(* CoDeSys 2.3.9.50 project: TcNcsample PTPmove.pro *)
(* Libraries: STANDARD.LIB 5.6.98 12:03:02, TcBase.lib 14.5.09 12:14:08, TcSystem.lib 7.6.16 11:01:22, TcNC.lib 10.10.08 17:55:34, TcMC.lib 27.7.15 08:51:38, TcBaseMath.lib 27.7.04 12:07:56, TcMath.lib 23.9.04 15:15:30 *)

(* Task configuration *)
TASK Standard (PRIORITY := 0, INTERVAL := T#10ms);
	MAIN
END_TASK

(* Global variable list: Global_Variables *)
VAR_GLOBAL
	(* =====================================================	*)
	(* NC · cyclical interface								*)
	(* =====================================================	*)

	PlcToNc AT %Q*	: PLCTONC_AXLESTRUCT;
	NcToPlc AT %I*	: NCTOPLC_AXLESTRUCT;
END_VAR

(* Global variable list: TwinCAT_Configuration *)
(* Generated automatically by TwinCAT - (read only) *)
VAR_CONFIG
	.PlcToNc AT %QB0 : PLCTONC_AXLESTRUCT;	(*  ~ {LinkedWith:TINC^NC-Task 1 SAF^Axes^Axis 1^Inputs^Axis 1_FromPlc} *)
	.NcToPlc AT %IB0 : NCTOPLC_AXLESTRUCT;	(*  ~ {LinkedWith:TINC^NC-Task 1 SAF^Axes^Axis 1^Outputs^Axis 1_ToPlc} *)
END_VAR

(* Data type *)
TYPE MoveState_t :
 (
	MOVESTATE_INIT,
	MOVESTATE_FORWARD,
	MOVESTATE_BACKWARDS
 );
END_TYPE

(* POU MAIN, ST *)
PROGRAM MAIN
VAR
	Position: LREAL;
	StartAxis: BOOL;
	MoveAxis: MC_MoveAbsolute;
	MoveDone: BOOL;
	MoveAborted: BOOL;
	MoveError: BOOL;
	MoveErrorID: UDINT;
	state: MoveState_t;
END_VAR
	(* enable the axis *)
	AxisEnable;

	(* 	move the axis forward and backwards
	*)
	CASE state OF
		MOVESTATE_INIT :	(* initialisation *)
			StartAxis := FALSE;
			IF AxisEnable.Ready THEN
				state := MOVESTATE_FORWARD;
			END_IF

		MOVESTATE_FORWARD :	(* start to first position *)
			Position := 2000;
			StartAxis := TRUE;
			IF MoveDone THEN
				StartAxis := FALSE;
				state := MOVESTATE_BACKWARDS;
			END_IF

		MOVESTATE_BACKWARDS :	(* move back to initial position *)
			Position := 0;
			StartAxis := TRUE;
			IF MoveDone THEN
				StartAxis := FALSE;
				state := MOVESTATE_FORWARD;
			END_IF
	END_CASE

	MoveAction;	(* call the move function block *)



	xxxx
	yyyy
zzzzzgit
END_PROGRAM
ACTION MoveAction:
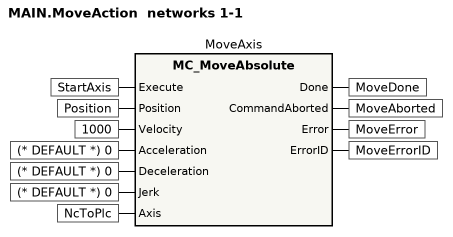
_FBD_ (* Function Block Diagram *)
NETWORK 1 (* Start axis using standard values FOR acceleration, deceleration AND jerk *)
	MoveAxis:MC_MoveAbsolute(Execute: StartAxis, Position: Position, Velocity: 1000, Acceleration: (* DEFAULT *) 0, Deceleration: (* DEFAULT *) 0, Jerk: (* DEFAULT *) 0, Axis: NcToPlc, CommandAborted => MoveAborted, Error => MoveError, ErrorID => MoveErrorID) => MoveDone
_END_FBD_
(* the same logic as Structured Text *)
(* Network 1: Start axis using standard values FOR acceleration, deceleration AND jerk *)
MoveAxis(Execute := StartAxis, Position := Position, Velocity := 1000, Acceleration := (* DEFAULT *) 0, Deceleration := (* DEFAULT *) 0, Jerk := (* DEFAULT *) 0, Axis := NcToPlc);
MoveAborted := MoveAxis.CommandAborted;
MoveError := MoveAxis.Error;
MoveErrorID := MoveAxis.ErrorID;
MoveDone := MoveAxis.Done;
END_ACTION

(* POU AxisEnable, FBD *)
PROGRAM AxisEnable
VAR_OUTPUT
	Ready: BOOL;
END_VAR
VAR
	Power: MC_Power;
	PowerError: BOOL;
	PowerErrorID: UDINT;
END_VAR
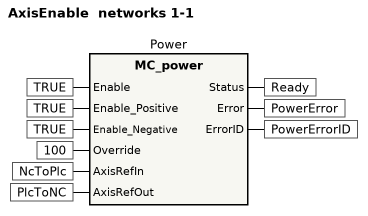
_FBD_ (* Function Block Diagram *)
NETWORK 1
	Power:MC_power(Enable: TRUE, Enable_Positive: TRUE, Enable_Negative: TRUE, Override: 100, AxisRefIn: NcToPlc, AxisRefOut: PlcToNC, Error => PowerError, ErrorID => PowerErrorID) => Ready
_END_FBD_
(* the same logic as Structured Text *)
(* Network 1 *)
Power(Enable := TRUE, Enable_Positive := TRUE, Enable_Negative := TRUE, Override := 100, AxisRefIn := NcToPlc, AxisRefOut := PlcToNC);
PowerError := Power.Error;
PowerErrorID := Power.ErrorID;
Ready := Power.Status;
END_PROGRAM
